// TIA Portal project "ArrayPlus_v000_000_004" (V16)
// v000.000.004: create Int[+].IsEmpty

(* hardware
DEVICE "S7-1200 station_1"  S7-1200 Station
   slot 0: "Rack_0"  S7-1200 Rack  Rack  V1.0
   slot 1: "PLC_1"  CPU 1212C DC/DC/DC  6ES7 212-1AE40-0XB0  V4.4
*)

// ===== PLC "PLC_1"  CPU 1212C DC/DC/DC =====

VAR_GLOBAL   // PLC tag table "Default tag table"
   "System_Byte" AT %MB1 : Byte;
   "FirstScan" AT %M1.0 : Bool;
   "DiagStatusUpdate" AT %M1.1 : Bool;
   "AlwaysTRUE" AT %M1.2 : Bool;
   "AlwaysFALSE" AT %M1.3 : Bool;
   "Clock_Byte" AT %MB0 : Byte;
   "Clock_10Hz" AT %M0.0 : Bool;
   "Clock_5Hz" AT %M0.1 : Bool;
   "Clock_2.5Hz" AT %M0.2 : Bool;
   "Clock_2Hz" AT %M0.3 : Bool;
   "Clock_1.25Hz" AT %M0.4 : Bool;
   "Clock_1Hz" AT %M0.5 : Bool;
   "Clock_0.625Hz" AT %M0.6 : Bool;
   "Clock_0.5Hz" AT %M0.7 : Bool;
END_VAR

TYPE "Int[+].UDT"
   STRUCT
      add : DInt;
      data : Array[0..4] of Int;
      length : DInt;
      remove : DInt := -1;
   END_STRUCT;
END_TYPE

FUNCTION "Int[+].IsFull" : Bool   // FC1, SCL
TITLE = Array Is Full
{ S7_Optimized_Access := 'TRUE' }
AUTHOR : Machado
FAMILY : Int[+]
VERSION : 0.1
// returns true if array is full
   VAR_INPUT
      buffer : "Int[+].UDT";
   END_VAR
   VAR_TEMP
      size : DInt;
   END_VAR
BEGIN
   #size := UDINT_TO_DINT("Int[].CountOfElements"(#buffer.data));
   IF #buffer.length = #size THEN
       #"Int[+].IsFull" := TRUE;
       RETURN;
   END_IF;
   #"Int[+].IsFull" := FALSE;
   RETURN;
END_FUNCTION

FUNCTION "Int[].CountOfElements" : UDInt   // FC2, SCL
{ S7_Optimized_Access := 'TRUE' }
VERSION : 0.1
   VAR_INPUT
      data : Variant;
   END_VAR
BEGIN
   #"Int[].CountOfElements" := CountOfElements(#data);
   RETURN;
END_FUNCTION

FUNCTION "Int[+].IsEmpty" : Bool   // FC3, SCL
TITLE = Int[+] Data Array Is Empty
{ S7_Optimized_Access := 'TRUE' }
AUTHOR : Machado
FAMILY : Int[+]
VERSION : 0.1
// returns true if array is empty
   VAR_INPUT
      buffer : "Int[+].UDT";
   END_VAR
BEGIN
   IF #buffer.length = 0 THEN
       #"Int[+].IsEmpty" := TRUE;
       RETURN;
   END_IF;
   #"Int[+].IsEmpty" := FALSE;
   RETURN;
END_FUNCTION

ORGANIZATION_BLOCK "Main"   // OB1, LAD, ProgramCycle
TITLE = "Main Program Sweep (Cycle)"
{ S7_Optimized_Access := 'TRUE' }
VERSION : 0.1
   VAR_INPUT
      Initial_Call : Bool;   // Initial call of this OB
      Remanence : Bool;   // =True, if remanent data are available
   END_VAR
BEGIN
END_ORGANIZATION_BLOCK